(* PLC project safety, BrAutomation SafeDESIGNER  5.8.0.0 *)
(* stored: companyURL http://www.br-automation.com, creationDateTime Tue Feb 11 10:07:14 2020 *)

PROGRAM Main
  VAR  (* added by the conversion: wires and edge detectors of the diagram *)
    _SAFEBOOL_TO_BOOL60_OUT : BOOL;
  END_VAR

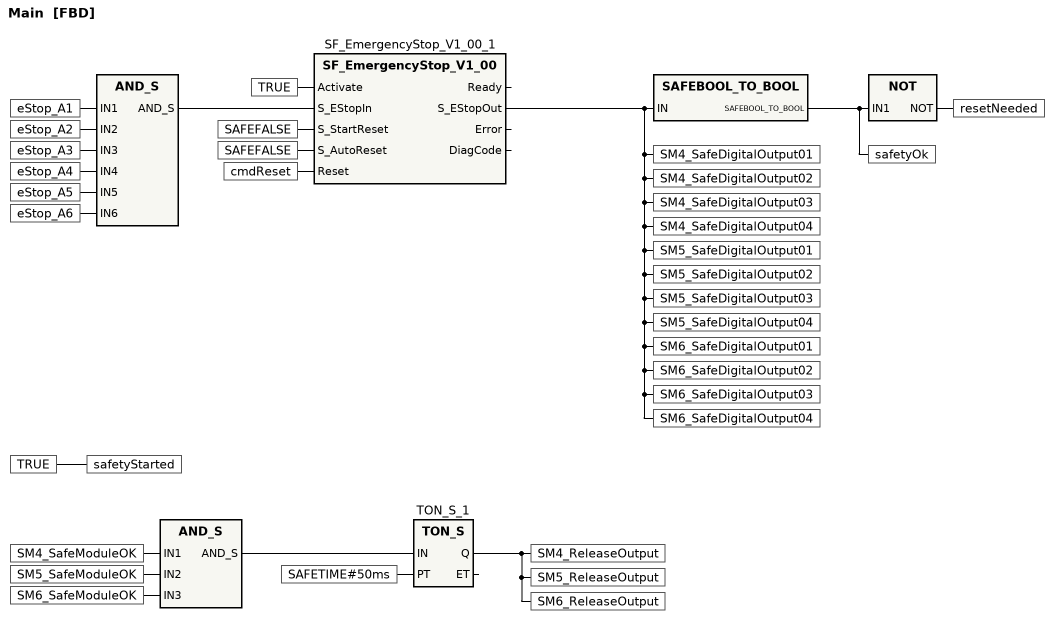
(* FBD diagram, written out as Structured Text *)
safetyStarted := TRUE;
SF_EmergencyStop_V1_00_1(Activate := TRUE, S_EStopIn := AND_S(eStop_A1, eStop_A2, eStop_A3, eStop_A4, eStop_A5, eStop_A6), S_StartReset := SAFEFALSE, S_AutoReset := SAFEFALSE, Reset := cmdReset);
_SAFEBOOL_TO_BOOL60_OUT := SAFEBOOL_TO_BOOL(SF_EmergencyStop_V1_00_1.S_EStopOut);
safetyOk := _SAFEBOOL_TO_BOOL60_OUT;
resetNeeded := NOT _SAFEBOOL_TO_BOOL60_OUT;
SM4_SafeDigitalOutput01 := SF_EmergencyStop_V1_00_1.S_EStopOut;
SM4_SafeDigitalOutput02 := SF_EmergencyStop_V1_00_1.S_EStopOut;
SM5_SafeDigitalOutput01 := SF_EmergencyStop_V1_00_1.S_EStopOut;
SM4_SafeDigitalOutput04 := SF_EmergencyStop_V1_00_1.S_EStopOut;
SM4_SafeDigitalOutput03 := SF_EmergencyStop_V1_00_1.S_EStopOut;
SM5_SafeDigitalOutput02 := SF_EmergencyStop_V1_00_1.S_EStopOut;
SM5_SafeDigitalOutput04 := SF_EmergencyStop_V1_00_1.S_EStopOut;
SM5_SafeDigitalOutput03 := SF_EmergencyStop_V1_00_1.S_EStopOut;
SM6_SafeDigitalOutput01 := SF_EmergencyStop_V1_00_1.S_EStopOut;
SM6_SafeDigitalOutput02 := SF_EmergencyStop_V1_00_1.S_EStopOut;
SM6_SafeDigitalOutput03 := SF_EmergencyStop_V1_00_1.S_EStopOut;
SM6_SafeDigitalOutput04 := SF_EmergencyStop_V1_00_1.S_EStopOut;
TON_S_1(IN := AND_S(SM4_SafeModuleOK, SM5_SafeModuleOK, SM6_SafeModuleOK), PT := SAFETIME#50ms);
SM5_ReleaseOutput := TON_S_1.Q;
SM4_ReleaseOutput := TON_S_1.Q;
SM6_ReleaseOutput := TON_S_1.Q;
END_PROGRAM
